// Mitsubishi GX Works2 project: PID_program_testing   PLC: FX2N/FX2NC

// task Task_01 (event FALSE, interval T#0.1s, priority 31): POU_01
// user libraries (not included): basic_lib

PROGRAM POU_01
VAR
  Paadrag : INT;
  ProcessValue : INT;
  PID_controller_1 : PID_controller;
  SetPoint : REAL;
  kp : REAL;
  ti : REAL;
  td : REAL;
  PID_controller_v2_1 : PID_controller_v2;
  MANAUTO : BOOL;
  manuelt_paadrag : INT;
  test_PV : INT;
  SampleTime : REAL;
  TON_1 : TON;
  SamplingstimeTracker_2 : SamplingstimeTracker;
  PID_controller_v3_1 : PID_controller_v3;
END_VAR
(* structured ladder/FBD written out as ST: instructions are called as NAME(EN, inputs, outputs); _pN, _eN, _tN stand for wires *)
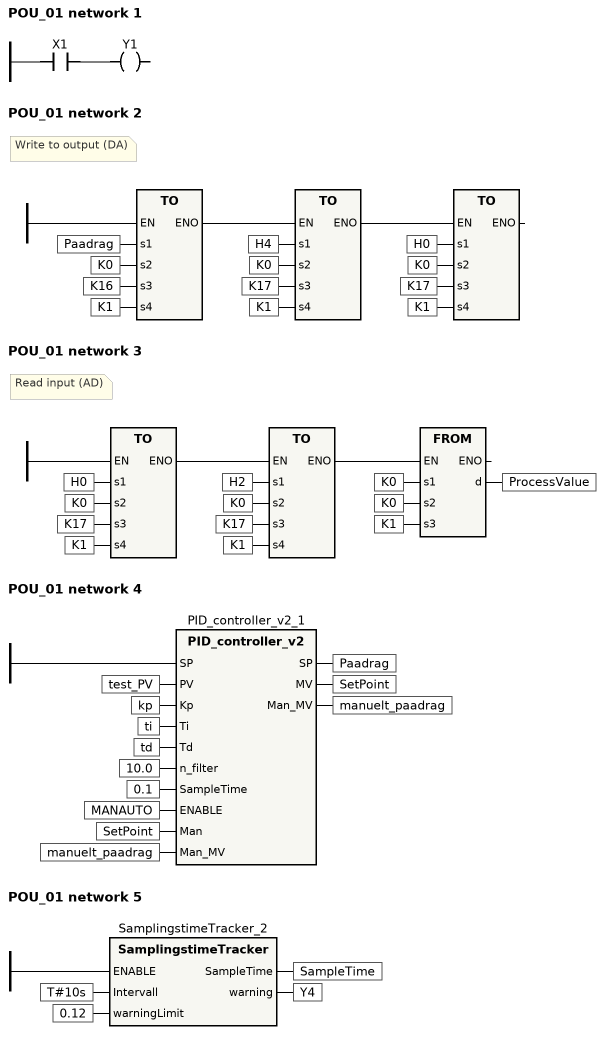
(* network 1 *)
Y1 := X1;
(* network 2 *)
(* Write to output (DA) *)
_e1 := TO(TRUE, Paadrag, K0, K16, K1);
_e2 := TO(_e1, H4, K0, K17, K1);
TO(_e2, H0, K0, K17, K1);
(* network 3 *)
(* Read input (AD) *)
_e1 := TO(TRUE, H0, K0, K17, K1);
_e2 := TO(_e1, H2, K0, K17, K1);
FROM(_e2, K0, K0, K1, ProcessValue);
(* network 4 *)
PID_controller_v2_1(SP := TRUE, PV := test_PV, Kp := kp, Ti := ti, Td := td, n_filter := 10.0, SampleTime := 0.1, ENABLE := MANAUTO, Man := SetPoint, Man_MV := manuelt_paadrag, MV => SetPoint);
Paadrag := PID_controller_v2_1.SP;
manuelt_paadrag := PID_controller_v2_1.Man_MV;
(* network 5 *)
SamplingstimeTracker_2(ENABLE := TRUE, Intervall := T#10s, warningLimit := 0.12, SampleTime => SampleTime, warning => Y4);
END_PROGRAM

FUNCTION_BLOCK PID_controller
VAR_INPUT
  SP : REAL;  (* Reference / Setpoint *)
  PV : INT;  (* Process Value *)
  Kp : REAL;  (* Proportional Gain *)
  Ti : REAL;  (* Integration Time *)
  Td : REAL;  (* Deviation Time *)
  n_filter : REAL;  (* Adjusting for filterconstant *)
  SampleTime : REAL;  (* In Seconds *)
END_VAR
VAR_OUTPUT
  MV : INT;  (* Modulated Value *)
END_VAR
VAR
  P_gain : REAL;
  I_gain : REAL;
  D_gain : REAL;
  Aa : REAL;  (* temporary variable *)
  Bb : REAL;  (* temporary variable *)
END_VAR
VAR CONSTANT
  MIN_INPUT : REAL;  (* These 4 constants are for satuating input and output *)
  MAX_INPUT : REAL := 255.0;  (* OBS: Variables may overflow if these values are too high / low *)
  MIN_OUTPUT : INT := -255;
  MAX_OUTPUT : INT := 255;
END_VAR
VAR
  Dev : REAL;  (* Deviation *)
END_VAR
VAR_INPUT
  ENABLE : BOOL;  (* Activate PID-block *)
END_VAR
VAR
  Dev_prev : REAL;  (* Previous value of Deviation *)
  PV_prev : REAL;  (* Previous value of Process Value *)
  I_gain_prev : REAL;  (* Previous value of I_gain *)
  D_gain_prev : REAL;  (* Previous value of D_gain *)
  PV_float : REAL;  (* Deviation *)
END_VAR
(*
		Had to rename variables in GX-works in order to avoid errors.
		
		Inputs:
			SP 		- 		reference / Setpoint
			PV 		- 		Process Value
			Kp  		- 		Propotional Gain
			Ti 		- 		Integration time
			Td  		- 		Derivation time
			n_filter- 		Adjusting the filter constant 	tau = Td / n
		
		Outputs:
			MV 		- 		Modulated Value
		
		Equations:
	 		MV			= P_gain  +  I_gain  +  D_gain
	 		P_gain	= Kp * e[k]
	 		I_gain	= KpT/(Ti*2) 	* 	(e[k] + e[k-1]) 		+		i[k-1] 	
	 		D_gain	= 2KpTd/(2) 	* 	(y[k]  -  y[k-1]) 		+		(2tau - T)/(2tau + T) * d[k-1]
*)

IF ENABLE = 0 THEN
	MV := 0;
ELSE 		
	(* 		Saturate input  		*)
	Aa := SP;  								(* Store to temporary variable for 2 reasons: 	1. Cant write new value to an input. *) 		
	FLT(1, PV, PV_float);			(* 																			  	2. Store space BY limiting number OF local variable definitions. *)
	IF Aa < MIN_INPUT THEN
		Aa := MIN_INPUT;
	ELSIF Aa > MAX_INPUT THEN
		Aa := MAX_INPUT;
	END_IF;
	
	IF PV_float < MIN_INPUT THEN
		PV_float := MIN_INPUT;
	ELSIF PV_float > MAX_INPUT THEN
		PV_float := MAX_INPUT;
	END_IF;

	(* 		Calculate deviation (avvik)	*)					
	Dev := Aa - PV_float;
	
	(* 		Calculate D 	*)
	Aa 			:= 2.0*Kp*Td / (2.0*(Td/n_filter)+ SampleTime);
	Bb 			:= (2.0*(Td/n_filter)- SampleTime) / (2.0*(Td/n_filter)+ SampleTime);
	D_gain 	:= Aa * ( PV_float - PV_prev ) + Bb * D_gain_prev;
	
	(* 		Calculate P 	*)
	P_gain 	:= Dev * Kp;
	
	(* 		Calculate I 		*)
	IF Ti = 0.0 THEN 			(* I_gain can be deactivated by setting Ti to 0. *)
		I_gain := 0.0;
	ELSE 
		Aa 		:= Kp * SampleTime / (2.0 * Ti);
		I_gain := Aa * (Dev + Dev_prev) + I_gain_prev;
	END_IF;
	
	(* Write to output*)
	INT(1, (P_gain + I_gain + D_gain), MV);
	
	(* Saturate output and check for windup *)
	IF MV < MIN_OUTPUT THEN 						(* Negative Saturation *)
		IF Dev < 0.0 THEN 										(* Antiwindup *)
			I_gain := I_gain_prev;
		END_IF;
		MV := MIN_OUTPUT;
	ELSIF MV > MAX_OUTPUT THEN 			(* Positive Saturation *)
		IF Dev > 0.0 THEN 										(* Antiwindup *)
			I_gain := I_gain_prev;
		END_IF;
		MV := MAX_OUTPUT;
	END_IF;
	
	(* Update previous values *)
	Dev_prev 		:= Dev;
	PV_prev 		:= PV_float;
	I_gain_prev 	:= I_gain;
	D_gain_prev 	:= D_gain; 
END_IF;
END_FUNCTION_BLOCK

FUNCTION_BLOCK PID_controller_v2
VAR_IN_OUT
  SP : REAL;  (* Reference / Setpoint *)
END_VAR
VAR_INPUT
  PV : INT;  (* Process Value *)
  Kp : REAL;  (* Proportional Gain *)
  Ti : REAL;  (* Integration Time *)
  Td : REAL;  (* Deviation Time *)
  n_filter : REAL;  (* Adjusting for filterconstant *)
  SampleTime : REAL;  (* In Seconds *)
END_VAR
VAR_OUTPUT
  MV : INT;  (* Modulated Value *)
END_VAR
VAR
  P_gain : REAL;
  I_gain : REAL;
  D_gain : REAL;
  Aa : REAL;  (* temporary variable *)
  Bb : REAL;  (* temporary variable *)
END_VAR
VAR CONSTANT
  MIN_INPUT : REAL;  (* These 4 constants are for satuating input and output *)
  MAX_INPUT : REAL := 255.0;  (* OBS: Variables may overflow if these values are too high / low *)
  MIN_OUTPUT : INT := -255;
  MAX_OUTPUT : INT := 255;
END_VAR
VAR
  Dev : REAL;  (* Deviation *)
END_VAR
VAR_INPUT
  ENABLE : BOOL;  (* Activate PID-block *)
END_VAR
VAR
  Dev_prev : REAL;  (* Previous value of Deviation *)
  PV_prev : REAL;  (* Previous value of Process Value *)
  I_gain_prev : REAL;  (* Previous value of I_gain *)
  D_gain_prev : REAL;  (* Previous value of D_gain *)
  PV_float : REAL;  (* Deviation *)
END_VAR
VAR_INPUT
  Man : BOOL;  (* Manuell/Auto. 1 = Man, 0 = Auto *)
END_VAR
VAR_IN_OUT
  Man_MV : INT;  (* Output is set to this value when in Manuell-mode *)
END_VAR
VAR
  ManAuto_flag : BOOL;  (* Tracks current state. 1 == Man. 0 == Auto *)
END_VAR
(*
		Had to rename variables in GX-works in order to avoid errors.
		
		Inputs:
			SP 		- 		reference / Setpoint
			PV 		- 		Process Value
			Kp  		- 		Propotional Gain
			Ti 		- 		Integration time
			Td  		- 		Derivation time
			n_filter- 		Adjusting the filter constant 	tau = Td / n
		
		Outputs:
			MV 		- 		Modulated Value
		
		Equations:
	 		MV			= P_gain  +  I_gain  +  D_gain
	 		P_gain	= Kp * e[k]
	 		I_gain		= KpT/(Ti*2) 	* 	(e[k] + e[k-1]) 		+		i[k-1] 	
	 		D_gain	= 2KpTd/(2) 	* 	(y[k]  -  y[k-1]) 		+		(2tau - T)/(2tau + T) * d[k-1]
*)

IF ENABLE = 0 THEN
	MV := 0;
ELSE 		
	IF NOT MAN THEN 			(* We're in AUTO *)
		
		(* 		Saturate input  		*)
		Aa := SP;  								(* Store to temporary variable for 2 reasons: 	1. Cant write new value to an input. *) 		
		FLT(1, PV, PV_float);			(* 																			  	2. Store space BY limiting number OF local variable definitions. *)
		IF Aa < MIN_INPUT THEN
			Aa := MIN_INPUT;
		ELSIF Aa > MAX_INPUT THEN
			Aa := MAX_INPUT;
		END_IF;
		
		IF PV_float < MIN_INPUT THEN
			PV_float := MIN_INPUT;
		ELSIF PV_float > MAX_INPUT THEN
			PV_float := MAX_INPUT;
		END_IF;
	
		(* 		Calculate deviation (avvik)	*)					
		Dev := Aa - PV_float;
		
		(* 		Calculate D 	*)
		Aa 			:= 2.0*Kp*Td / (2.0*(Td/n_filter)+ SampleTime);
		Bb 			:= (2.0*(Td/n_filter)- SampleTime) / (2.0*(Td/n_filter)+ SampleTime);
		D_gain 	:= Aa * ( PV_float - PV_prev ) + Bb * D_gain_prev;
		
		(* 		Calculate P 	*)
		P_gain 	:= Dev * Kp;
		
		(* 		This prevents huge jumps in MV when switching from MAN to AUTO	 *)
		IF ManAuto_flag THEN
			FLT(1, Man_MV, I_gain);	
			ManAuto_flag 	:= FALSE;
		ELSE 
			
			(* 		Calculate I 		*)
			IF Ti = 0.0 THEN 			(* I_gain can be deactivated by setting Ti to 0. *)
				I_gain := 0.0;
			ELSE 
				Aa 		:= Kp * SampleTime / (2.0 * Ti);
				I_gain := Aa * (Dev + Dev_prev) + I_gain_prev;
			END_IF;
				
		END_IF;
		
		(* Write to output*)
		INT(1, (P_gain + I_gain + D_gain), MV);
		
		(* Saturate output and check for windup *)
		IF MV < MIN_OUTPUT THEN 						(* Negative Saturation *)
			IF Dev < 0.0 THEN 										(* Antiwindup *)
				I_gain := I_gain_prev;
			END_IF;
			MV := MIN_OUTPUT;
		ELSIF MV > MAX_OUTPUT THEN 				(* Positive Saturation *)
			IF Dev > 0.0 THEN 										(* Antiwindup *)
				I_gain := I_gain_prev;
			END_IF;
			MV := MAX_OUTPUT;
		END_IF;
		
		(* Update previous values *)
		Dev_prev 		:= Dev;
		PV_prev 		:= PV_float;
		I_gain_prev 	:= I_gain;
		D_gain_prev 	:= D_gain; 
		
		ELSE  			(* We're in MAN *)
			(* This prevents huge jumps  when switching from AUTO to MAN. It is both input and output - meaning that Man_MV on HMI should be read-write *)
			IF NOT ManAuto_flag THEN
				INT(1, (P_gain + I_gain + D_gain), Man_MV);
				ManAuto_flag := TRUE;
			END_IF;
			MV := Man_MV;
			FLT(1, PV, SP);			(* Continouly update Setpoint while in MAN mode *)
			
			(* Saturate both values *)
			IF MV > MAX_OUTPUT THEN
				MV 			 := MAX_OUTPUT;
				Man_MV := MAX_OUTPUT;
			ELSIF MV < MIN_OUTPUT THEN
				MV 			 := MIN_OUTPUT;
				Man_MV := MIN_OUTPUT;
			END_IF;
				
		END_IF;
END_IF;
END_FUNCTION_BLOCK

FUNCTION_BLOCK SamplingstimeTracker
VAR_INPUT
  ENABLE : BOOL;  (* Activate block *)
  Intervall : TIME;  (* Time between each caluclation *)
END_VAR
VAR_OUTPUT
  SampleTime : REAL;  (* In seconds *)
END_VAR
VAR
  counter : DINT;  (* Increments every cycle *)
  tonFlag : BOOL;
  tonCurrentTIme : TIME;
  time_DINT : DINT;  (* Temporary variable *)
  counter_FLT : REAL;  (* Temporary variable *)
  time_FLT : REAL;  (* Temporary variable *)
  TON_1 : TON;
END_VAR
VAR_INPUT
  warningLimit : REAL;  (* Used for output "warning" *)
END_VAR
VAR_OUTPUT
  warning : BOOL;  (* High if SampleTime > warningLimit *)
END_VAR
(*
	==== 		SampletimeTracker 		====
	

*)

IF ENABLE THEN
	DINC(1, counter);
	TON_1(IN:=1, PT:=Intervall, Q:=tonFlag , ET:=tonCurrentTIme); 			(* Start timer *)
	
	IF tonFlag THEN 
		(* Calculate SampleTime*)
		 time_DINT := TIME_TO_DINT(tonCurrentTIme); 			(* Milliseconds *)
		DFLT(1, time_DINT, time_FLT); 								
		DFLT(1, counter, counter_FLT);
		SampleTime := time_FLT/(counter_FLT*1000.0);
		
		(* Reset variables *)
		TON_1(IN:=0, PT:=Intervall, Q:=tonFlag , ET:=tonCurrentTIme);  		(* Reset timer *)
		counter := 0; 
	END_IF;
	
	(* 	Warning / Alarm *)
	IF SampleTime > warningLimit THEN
		warning := TRUE;	
	END_IF;
	
END_IF;
END_FUNCTION_BLOCK

FUNCTION_BLOCK PID_controller_v3
VAR_INPUT
  SP : REAL;  (* Reference / Setpoint *)
  PV : INT;  (* Process Value *)
  Kp : REAL;  (* Proportional Gain *)
  Ti : REAL;  (* Integration Time *)
  Td : REAL;  (* Deviation Time *)
  n_filter : REAL;  (* Adjusting for filterconstant *)
  SampleTime : REAL;  (* In Seconds *)
END_VAR
VAR_OUTPUT
  MV : INT;  (* Modulated Value *)
END_VAR
VAR
  P_gain : REAL;
  I_gain : REAL;
  D_gain : REAL;
  Aa : REAL;  (* temporary variable *)
  Bb : REAL;  (* temporary variable *)
END_VAR
VAR CONSTANT
  MIN_INPUT : REAL;  (* These 4 constants are for satuating input and output *)
  MAX_INPUT : REAL := 255.0;  (* OBS: Variables may overflow if these values are too high / low *)
  MIN_OUTPUT : INT := -255;
  MAX_OUTPUT : INT := 255;
END_VAR
VAR
  Dev : REAL;  (* Deviation *)
END_VAR
VAR_INPUT
  ENABLE : BOOL;  (* Activate PID-block *)
END_VAR
VAR
  Dev_prev : REAL;  (* Previous value of Deviation *)
  PV_prev : REAL;  (* Previous value of Process Value *)
  I_gain_prev : REAL;  (* Previous value of I_gain *)
  D_gain_prev : REAL;  (* Previous value of D_gain *)
  PV_float : REAL;  (* Process Value (type float) *)
END_VAR
VAR_INPUT
  Tracking : INT;  (* Tracking *)
END_VAR
(*
		Had to rename variables in GX-works in order to avoid errors.
		
		Inputs:
			SP 				- 		reference / Setpoint
			PV 				- 		Process Value
			Kp  				- 		Propotional Gain
			Ti 				- 		Integration time
			Td  				- 		Derivation time
			n_filter		- 		Adjusting the filter constant 	tau = Td / n
			Tracking 	- 		Tracking input. Used when using more than 1 controller in paralell.
		
		Outputs:
			MV 		- 		Modulated Value
		
		Equations:
	 		MV			= P_gain  +  I_gain  +  D_gain
	 		P_gain	= Kp * e[k]
	 		I_gain		= KpT/(Ti*2) 	* 	(e[k] + e[k-1]) 		+		i[k-1] 	
	 		D_gain	= 2KpTd/(2) 	* 	(y[k]  -  y[k-1]) 		+		(2tau - T)/(2tau + T) * d[k-1]
	 		
	 	Tracking:
			I_gain on the controller can be deactivated by setting Ti = 0.0.
			In order for Tracking to work - Ti needs to be higher than 0.0.
*)

IF ENABLE = 0 THEN
	MV := 0;
ELSE 		
	(* 		Saturate input  		*)
	Aa := SP;  								(* Store to temporary variable for 2 reasons: 	1. Cant write new value to an input. *) 		
	FLT(1, PV, PV_float);			(* 																		2. Store space BY limiting number OF local variable definitions. *)
	IF Aa < MIN_INPUT THEN
		Aa := MIN_INPUT;
	ELSIF Aa > MAX_INPUT THEN
		Aa := MAX_INPUT;
	END_IF;
	
	IF PV_float < MIN_INPUT THEN
		PV_float := MIN_INPUT;
	ELSIF PV_float > MAX_INPUT THEN
		PV_float := MAX_INPUT;
	END_IF;

	(* 		Calculate deviation (avvik)	*)					
	Dev := Aa - PV_float;
	
	(* 		Calculate D 	*)
	Aa 			:= 2.0*Kp*Td / (2.0*(Td/n_filter)+ SampleTime);
	Bb 			:= (2.0*(Td/n_filter)- SampleTime) / (2.0*(Td/n_filter)+ SampleTime);
	D_gain 	:= Aa * ( PV_float - PV_prev ) + Bb * D_gain_prev;
	
	(* 		Calculate P 	*)
	P_gain 	:= Dev * Kp;
	
	(* 		Calculate I 		*)
	IF Ti = 0.0 THEN 			(* I_gain can be deactivated by setting Ti to 0. *)
		I_gain := 0.0;
	ELSE 
		IF MV = Tracking THEN 	(* Note that this MV is from the last cycle and has not been updated YET *)
			Aa 		 := Kp * SampleTime / (2.0 * Ti);
			I_gain := Aa * (Dev + Dev_prev) + I_gain_prev;
		ELSE
			(*This controller is not in control. Activate Tracking *)
			FLT(1, Tracking, Aa);
			I_gain := Aa - P_gain - D_gain;	
		END_IF;
	END_IF;
	
	(* Write to output*)
	INT(1, (P_gain + I_gain + D_gain), MV);
	
	(* Saturate output and check for windup *)
	IF MV < MIN_OUTPUT THEN 						(* Negative Saturation *)
		IF Dev < 0.0 THEN 										(* Antiwindup *)
			I_gain := I_gain_prev;
		END_IF;
		MV := MIN_OUTPUT;
	ELSIF MV > MAX_OUTPUT THEN 			(* Positive Saturation *)
		IF Dev > 0.0 THEN 										(* Antiwindup *)
			I_gain := I_gain_prev;
		END_IF;
		MV := MAX_OUTPUT;
	END_IF;
	
	(* Update previous values *)
	Dev_prev 		:= Dev;
	PV_prev 			:= PV_float;
	I_gain_prev 	:= I_gain;
	D_gain_prev 	:= D_gain; 
END_IF;
END_FUNCTION_BLOCK
